{attribute 'qualified_only'}
VAR_GLOBAL
	SW_00	AT%IX0.0	:BOOL;
	SW_01	AT%IX0.1	:BOOL;
	SW_02	AT%IX0.2	:BOOL;
	EMS  	AT%IX0.3	:BOOL;
	CS_01	AT%IX0.4	:BOOL;
	CS_02	AT%IX0.5	:BOOL;
	CS_03	AT%IX0.6	:BOOL;
	CS_04	AT%IX0.7	:BOOL;
	CS_05	AT%IX1.0	:BOOL;
	CS_06	AT%IX1.1	:BOOL;
	CS_07	AT%IX1.2	:BOOL;
	CS_08	AT%IX1.3	:BOOL;
	S_01	AT%IX1.4	:BOOL;
	S_02	AT%IX1.5	:BOOL;
	S_03	AT%IX1.6	:BOOL;
	S_04	AT%IX1.7	:BOOL;
	
	SOL_01	AT%QX0.0	:BOOL;
	SOL_02	AT%QX0.1	:BOOL;
	SOL_03	AT%QX0.2	:BOOL;
	SOL_04	AT%QX0.3	:BOOL;
	SOL_05	AT%QX0.4	:BOOL;
	M_01	AT%QX0.5	:BOOL;
	M_02	AT%QX0.6	:BOOL;
	L_01	AT%QX0.7	:BOOL;
	L_02	AT%QX1.0	:BOOL;
	L_03	AT%QX1.1	:BOOL;
	CT		AT%QX1.2	:BOOL;
	
END_VAR

(* stored: Version 1.1.0.1, ProductVersion 3.1.4024.6
   GVL GVL: Id {f0692d3a-e688-46af-9fcd-56b8a7d83856} *)
